KUKA KRL program: wkz7_off.src, wkz7_off.dat

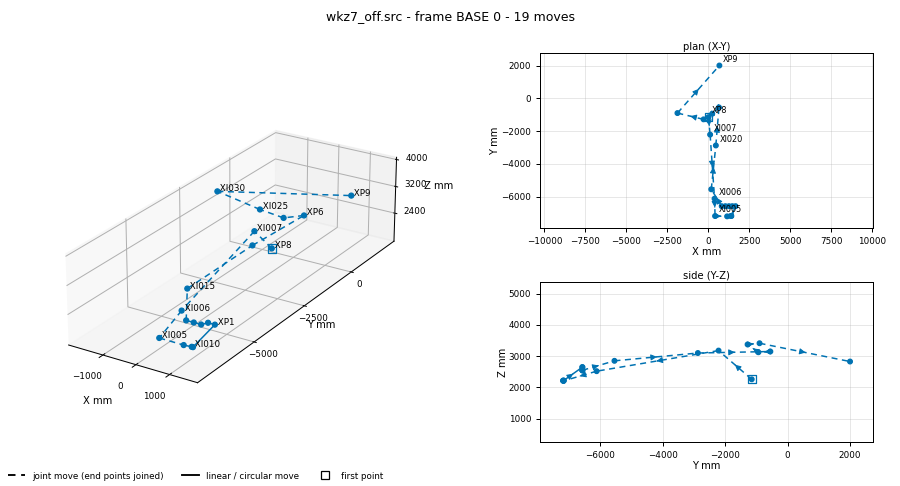
[picture p0: tool path of wkz7_off.src in frame BASE 0, 19 of 19 moves have a stored position in this frame; points joined in program order, loops and branches not executed]
--- wkz7_off.src ---
&ACCESS RVO7
&REL 553
&COMMENT Pega Gripper Axor GeoBox
&PARAM DISKPATH = KRC:\R1\Program
&PARAM TEMPLATE = C:\KRC\Roboter\Template\vorgabe
&PARAM EDITMASK = *
DEF WKZ7_OFF ( )
;FOLD INI
  ;FOLD BASISTECH INI
    GLOBAL INTERRUPT DECL 3 WHEN $STOPMESS==TRUE DO IR_STOPM ( )
    INTERRUPT ON 3
    BAS (#INITMOV,0)
  ;ENDFOLD (BASISTECH INI)
;FOLD GRIPPERTECH INI
USER_GRP(0,DUMMY,DUMMY,GDEFAULT)
;ENDFOLD (GRIPPERTECH INI)
  ;FOLD USER INI
    ;Make your modifications here

  ;ENDFOLD (USER INI)
;ENDFOLD (INI)

; Caracterizacao dos meios de producao:
; Changes: Pega Gripper na GeoBox
; Versao Atual:27/08/2015
; Name: P13.050-R2

chk_w8_wechs_ok ( )       ; CHECK TOOL CHANGE

; LIGA INTERLOCK 5 C/ R5
;FOLD Collision.Monitoring_5_On ;%{PE}%MKUKATPUSER
COLLSTOP( 5, 1 ) ;not Interrupt-Controlled
;ENDFOLD

;FOLD PTP P8 CONT Vel=100 % PDAT8 Tool[7]:Garra AXOR Base[0];%{PE}%R 8.2.20,%MKUKATPBASIS,%CMOVE,%VPTP,%P 1:PTP, 2:P8, 3:C_DIS, 5:100, 7:PDAT8
$BWDSTART=FALSE
PDAT_ACT=PPDAT8
FDAT_ACT=FP8
BAS(#PTP_PARAMS,100)
PTP XP8 C_DIS
;ENDFOLD
;FOLD PTP l007 CONT Vel=100 % P_OLP10 Tool[7]:Garra AXOR Base[0];%{PE}%R 8.2.20,%MKUKATPBASIS,%CMOVE,%VPTP,%P 1:PTP, 2:l007, 3:C_DIS, 5:100, 7:P_OLP10
$BWDSTART=FALSE
PDAT_ACT=PP_OLP10
FDAT_ACT=Fl007
BAS(#PTP_PARAMS,100)
PTP Xl007 C_DIS
;ENDFOLD
;FOLD PTP l006 CONT Vel=100 % P_OLP9 Tool[7]:Garra AXOR Base[0];%{PE}%R 8.2.20,%MKUKATPBASIS,%CMOVE,%VPTP,%P 1:PTP, 2:l006, 3:C_DIS, 5:100, 7:P_OLP9
$BWDSTART=FALSE
PDAT_ACT=PP_OLP9
FDAT_ACT=Fl006
BAS(#PTP_PARAMS,100)
PTP Xl006 C_DIS
;ENDFOLD
;FOLD PTP l005 CONT Vel=100 % P_OLP2 Tool[7]:Garra AXOR Base[0];%{PE}%R 8.2.20,%MKUKATPBASIS,%CMOVE,%VPTP,%P 1:PTP, 2:l005, 3:C_DIS, 5:100, 7:P_OLP2
$BWDSTART=FALSE
PDAT_ACT=PP_OLP2
FDAT_ACT=Fl005
BAS(#PTP_PARAMS,100)
PTP Xl005 C_DIS
;ENDFOLD
;FOLD PTP P10 Vel=100 % PDAT10 Tool[8]:Tool Changer Base[0];%{PE}%R 8.2.20,%MKUKATPBASIS,%CMOVE,%VPTP,%P 1:PTP, 2:P10, 3:, 5:100, 7:PDAT10
$BWDSTART=FALSE
PDAT_ACT=PPDAT10
FDAT_ACT=FP10
BAS(#PTP_PARAMS,100)
PTP XP10
;ENDFOLD

;FOLD OUT 3378 'Lib. p/ retirar Gripper GeoBox' State=TRUE ;%{PE}%R 8.2.20,%MKUKATPBASIS,%COUT,%VOUTX,%P 2:3378, 3:Lib. p/ retirar Gripper GeoBox, 5:TRUE, 6:
$OUT[3378]=TRUE
;ENDFOLD
;FOLD WAIT FOR ( IN 3378 'Lib. p/ retirar Gripper GeoBox' );%{PE}%R 8.2.20,%MKUKATPBASIS,%CEXT_WAIT_FOR,%VEXT_WAIT_FOR,%P 2:, 4:, 5:$IN, 6:3378, 7:Lib. p/ retirar Gripper GeoBox, 9:
WAIT FOR  ( $IN[3378] )
;ENDFOLD
;FOLD OUT 3378 'Lib. p/ retirar Gripper GeoBox' State=FALSE ;%{PE}%R 8.2.20,%MKUKATPBASIS,%COUT,%VOUTX,%P 2:3378, 3:Lib. p/ retirar Gripper GeoBox, 5:FALSE, 6:
$OUT[3378]=FALSE
;ENDFOLD
;FOLD OUT 3348 'Fora area GEOBOX' State=FALSE ;%{PE}%R 8.2.20,%MKUKATPBASIS,%COUT,%VOUTX,%P 2:3348, 3:Fora area GEOBOX, 5:FALSE, 6:
$OUT[3348]=FALSE
;ENDFOLD


;FOLD LIN l010 Vel=1 m/s CPDAT4 Tool[8]:Tool Changer Base[0];%{PE}%R 8.2.20,%MKUKATPBASIS,%CMOVE,%VLIN,%P 1:LIN, 2:l010, 3:, 5:1, 7:CPDAT4
$BWDSTART=FALSE
LDAT_ACT=LCPDAT4
FDAT_ACT=Fl010
BAS(#CP_PARAMS,1)
LIN Xl010
;ENDFOLD

;FOLD OUT 224 'Bloquear MPS' State=FALSE ;%{PE}%R 8.2.20,%MKUKATPBASIS,%COUT,%VOUTX,%P 2:224, 3:Bloquear MPS, 5:FALSE, 6:
$OUT[224]=FALSE
;ENDFOLD
;FOLD OUT 223 'Desbloquear MPS' State=TRUE ;%{PE}%R 8.2.20,%MKUKATPBASIS,%COUT,%VOUTX,%P 2:223, 3:Desbloquear MPS, 5:TRUE, 6:
$OUT[223]=TRUE
;ENDFOLD
;FOLD WAIT FOR ( IN 217 'MPS Destravado' );%{PE}%R 8.2.20,%MKUKATPBASIS,%CEXT_WAIT_FOR,%VEXT_WAIT_FOR,%P 2:, 4:, 5:$IN, 6:217, 7:MPS Destravado, 9:
WAIT FOR  ( $IN[217] )
;ENDFOLD
;FOLD WAIT FOR NOT ( IN 221 'MPS Travado' );%{PE}%R 8.2.20,%MKUKATPBASIS,%CEXT_WAIT_FOR,%VEXT_WAIT_FOR,%P 2:NOT, 4:, 5:$IN, 6:221, 7:MPS Travado, 9:
WAIT FOR  NOT ( $IN[221] )
;ENDFOLD

;FOLD ; Posicao de Pega Gripper AXOR na Geobox;%{PE}%R 8.2.20,%MKUKATPBASIS,%CCOMMENT,%VNORMAL,%P 2:Posicao de Pega Gripper  AXOR na Geobox
;ENDFOLD
;FOLD LIN P_PE11 Vel=1 m/s CPDAT6 Tool[8]:Tool Changer Base[0];%{PE}%R 8.2.20,%MKUKATPBASIS,%CMOVE,%VLIN,%P 1:LIN, 2:P_PE11, 3:, 5:1, 7:CPDAT6
$BWDSTART=FALSE
LDAT_ACT=LCPDAT6
FDAT_ACT=FP_PE11
BAS(#CP_PARAMS,1)
LIN XP_PE11
;ENDFOLD

;FOLD WAIT FOR ( IN 219 'Posicao p/ Acoplamento OK' );%{PE}%R 8.2.20,%MKUKATPBASIS,%CEXT_WAIT_FOR,%VEXT_WAIT_FOR,%P 2:, 4:, 5:$IN, 6:219, 7:Posicao p/ Acoplamento OK, 9:
WAIT FOR  ( $IN[219] )
;ENDFOLD
;FOLD OUT 223 'Desbloquear MPS' State=FALSE ;%{PE}%R 8.2.20,%MKUKATPBASIS,%COUT,%VOUTX,%P 2:223, 3:Desbloquear MPS, 5:FALSE, 6:
$OUT[223]=FALSE
;ENDFOLD
;FOLD OUT 224 'Bloquear MPS' State=TRUE ;%{PE}%R 8.2.20,%MKUKATPBASIS,%COUT,%VOUTX,%P 2:224, 3:Bloquear MPS, 5:TRUE, 6:
$OUT[224]=TRUE
;ENDFOLD
;FOLD WAIT FOR NOT ( IN 217 'MPS Destravado' );%{PE}%R 8.2.20,%MKUKATPBASIS,%CEXT_WAIT_FOR,%VEXT_WAIT_FOR,%P 2:NOT, 4:, 5:$IN, 6:217, 7:MPS Destravado, 9:
WAIT FOR  NOT ( $IN[217] )
;ENDFOLD
;FOLD WAIT FOR ( IN 221 'MPS Travado' );%{PE}%R 8.2.20,%MKUKATPBASIS,%CEXT_WAIT_FOR,%VEXT_WAIT_FOR,%P 2:, 4:, 5:$IN, 6:221, 7:MPS Travado, 9:
WAIT FOR  ( $IN[221] )
;ENDFOLD
;FOLD WAIT Time=0.5 sec;%{PE}%R 8.2.20,%MKUKATPBASIS,%CWAIT,%VWAIT,%P 3:0.5
WAIT SEC 0.5
;ENDFOLD
;FOLD IBUS ON SEGMENT_4;%{PE}%R 8.2.20,%MKUKATPBASIS,%CIBUS,%VMAP,%P 2:#ON, 3:4
$IBUS_ON=IBUS_SEGMENT[4]
$IBUS_OFF=0
;ENDFOLD
;FOLD WAIT Time=0.5 sec;%{PE}%R 8.2.20,%MKUKATPBASIS,%CWAIT,%VWAIT,%P 3:0.5
WAIT SEC 0.5
;ENDFOLD

;FOLD OUT 3379 'Lib. p/ sair c/ Gripper GeoBox' State=TRUE ;%{PE}%R 8.2.20,%MKUKATPBASIS,%COUT,%VOUTX,%P 2:3379, 3:Lib. p/ sair c/ Gripper GeoBox, 5:TRUE, 6:
$OUT[3379]=TRUE
;ENDFOLD

; ABRE GRAMPOS
;FOLD SET VACUO AXOR State=BLOW GDAT11;%{PE}%R 8.2.1,%MKUKATPGRP,%CGRP,%VGRP,%P 2:9, 4:2, 5:#NO, 6:GDAT11, 8:0, 10:0
H50(GRP,9,2,GGDAT11)
;ENDFOLD
;FOLD SET VACUO AXOR State=OFF GDAT12;%{PE}%R 8.2.1,%MKUKATPGRP,%CGRP,%VGRP,%P 2:9, 4:3, 5:#NO, 6:GDAT12, 8:0, 10:0
H50(GRP,9,3,GGDAT12)
;ENDFOLD
;FOLD SET Z2.1 RPS AXOR State=OPN GDAT25;%{PE}%R 8.2.1,%MKUKATPGRP,%CGRP,%VGRP,%P 2:10, 4:1, 5:#NO, 6:GDAT25, 8:0, 10:0
H50(GRP,10,1,GGDAT25)
;ENDFOLD
;FOLD SET Z4.1 GRP AXOR State=OPN GDAT13;%{PE}%R 8.2.1,%MKUKATPGRP,%CGRP,%VGRP,%P 2:12, 4:1, 5:#NO, 6:GDAT13, 8:0, 10:0
H50(GRP,12,1,GGDAT13)
;ENDFOLD
;FOLD SET Z5.1/2/3/4 GRP AXOR State=OPN GDAT16;%{PE}%R 8.2.1,%MKUKATPGRP,%CGRP,%VGRP,%P 2:13, 4:1, 5:#NO, 6:GDAT16, 8:0, 10:0
H50(GRP,13,1,GGDAT16)
;ENDFOLD
;FOLD SET Z6.1/2/3/4 GRP AXOR State=OPN GDAT17;%{PE}%R 8.2.1,%MKUKATPGRP,%CGRP,%VGRP,%P 2:14, 4:1, 5:#NO, 6:GDAT17, 8:0, 10:0
H50(GRP,14,1,GGDAT17)
;ENDFOLD
;FOLD SET Z7.1/2 GRP AXOR State=OPN GDAT18;%{PE}%R 8.2.1,%MKUKATPGRP,%CGRP,%VGRP,%P 2:15, 4:1, 5:#NO, 6:GDAT18, 8:0, 10:0
H50(GRP,15,1,GGDAT18)
;ENDFOLD

; VERIFICA GRAMPOS FECHADOS
chk_w7_rps2_opn( )
chk_w7_grp4_opn( )
chk_w7_grp5_opn( )
chk_w7_grp1_vacoff( )

; ABRE GRAMPO Z3.1 e VERIFICA
;FOLD SET Z3.1 GRP AXOR State=OPN GDAT26;%{PE}%R 8.2.1,%MKUKATPGRP,%CGRP,%VGRP,%P 2:11, 4:1, 5:#NO, 6:GDAT26, 8:0, 10:0
H50(GRP,11,1,GGDAT26)
;ENDFOLD
chk_w7_grp6_opn( )
chk_w7_grp7_opn( )
chk_w7_grp3_opn( )

;FOLD OUT 3379 'Solicita lib. p/ sair c/ Gripper GeoBox' State=TRUE ;%{PE}%R 8.2.20,%MKUKATPBASIS,%COUT,%VOUTX,%P 2:3379, 3:Solicita lib. p/ sair c/ Gripper GeoBox, 5:TRUE, 6:
$OUT[3379]=TRUE
;ENDFOLD
;FOLD WAIT FOR ( IN 3379 'Aguarda lib. p/ sair c/ Gripper GeoBox' );%{PE}%R 8.2.20,%MKUKATPBASIS,%CEXT_WAIT_FOR,%VEXT_WAIT_FOR,%P 2:, 4:, 5:$IN, 6:3379, 7:Aguarda lib. p/ sair c/ Gripper GeoBox, 9:
WAIT FOR  ( $IN[3379] )
;ENDFOLD
;FOLD OUT 3379 'Solicita lib. p/ sair c/ Gripper GeoBox' State=FALSE ;%{PE}%R 8.2.20,%MKUKATPBASIS,%COUT,%VOUTX,%P 2:3379, 3:Solicita lib. p/ sair c/ Gripper GeoBox, 5:FALSE, 6:
$OUT[3379]=FALSE
;ENDFOLD

;FOLD LIN P1 CONT Vel=1 m/s CPDAT2 Tool[7]:Garra AXOR Base[0];%{PE}%R 8.2.20,%MKUKATPBASIS,%CMOVE,%VLIN,%P 1:LIN, 2:P1, 3:C_DIS C_DIS, 5:1, 7:CPDAT2
$BWDSTART=FALSE
LDAT_ACT=LCPDAT2
FDAT_ACT=FP1
BAS(#CP_PARAMS,1)
LIN XP1 C_DIS C_DIS
;ENDFOLD
;FOLD LIN P3 CONT Vel=1 m/s CPDAT5 Tool[7]:Garra AXOR Base[0];%{PE}%R 8.2.20,%MKUKATPBASIS,%CMOVE,%VLIN,%P 1:LIN, 2:P3, 3:C_DIS C_DIS, 5:1, 7:CPDAT5
$BWDSTART=FALSE
LDAT_ACT=LCPDAT5
FDAT_ACT=FP3
BAS(#CP_PARAMS,1)
LIN XP3 C_DIS C_DIS
;ENDFOLD

;FOLD LIN P14 Vel=1 m/s CPDAT9 Tool[7]:Garra AXOR Base[0];%{PE}%R 8.2.20,%MKUKATPBASIS,%CMOVE,%VLIN,%P 1:LIN, 2:P14, 3:, 5:1, 7:CPDAT9
$BWDSTART=FALSE
LDAT_ACT=LCPDAT9
FDAT_ACT=FP14
BAS(#CP_PARAMS,1)
LIN XP14
;ENDFOLD

;FOLD PULSE 3335 'R2 retirou garra da Geo' State=TRUE Time=3 sec;%{PE}%R 8.2.20,%MKUKATPBASIS,%COUT,%VPULSE,%P 2:3335, 3:R2 retirou garra da Geo, 5:TRUE, 6:, 8:3
PULSE($OUT[3335], TRUE,3)
;ENDFOLD

;FOLD PTP P13 CONT Vel=100 % PDAT12 Tool[7]:Garra AXOR Base[0];%{PE}%R 8.2.20,%MKUKATPBASIS,%CMOVE,%VPTP,%P 1:PTP, 2:P13, 3:C_DIS, 5:100, 7:PDAT12
$BWDSTART=FALSE
PDAT_ACT=PPDAT12
FDAT_ACT=FP13
BAS(#PTP_PARAMS,100)
PTP XP13 C_DIS
;ENDFOLD

; DESLIGA INTERLOCK 5 C/ R5
;FOLD Collision.Monitoring_5_Off . ;%{PE}%MKUKATPUSER
COLLSTOP( 5, 2+0 )
;ENDFOLD

;FOLD PTP P11 CONT Vel=100 % PDAT13 Tool[7]:Garra AXOR Base[0];%{PE}%R 8.2.20,%MKUKATPBASIS,%CMOVE,%VPTP,%P 1:PTP, 2:P11, 3:C_DIS, 5:100, 7:PDAT13
$BWDSTART=FALSE
PDAT_ACT=PPDAT13
FDAT_ACT=FP11
BAS(#PTP_PARAMS,100)
PTP XP11 C_DIS
;ENDFOLD
;FOLD PTP l015 CONT Vel=100 % PDAT4 Tool[7]:Garra AXOR Base[0];%{PE}%R 8.2.20,%MKUKATPBASIS,%CMOVE,%VPTP,%P 1:PTP, 2:l015, 3:C_DIS, 5:100, 7:PDAT4
$BWDSTART=FALSE
PDAT_ACT=PPDAT4
FDAT_ACT=Fl015
BAS(#PTP_PARAMS,100)
PTP Xl015 C_DIS
;ENDFOLD
;FOLD PTP l020 CONT Vel=100 % P_OLP4 Tool[7]:Garra AXOR Base[0];%{PE}%R 8.2.20,%MKUKATPBASIS,%CMOVE,%VPTP,%P 1:PTP, 2:l020, 3:C_DIS, 5:100, 7:P_OLP4
$BWDSTART=FALSE
PDAT_ACT=PP_OLP4
FDAT_ACT=Fl020
BAS(#PTP_PARAMS,100)
PTP Xl020 C_DIS
;ENDFOLD
;FOLD PTP P6 CONT Vel=100 % PDAT6 Tool[7]:Garra AXOR Base[0];%{PE}%R 8.2.20,%MKUKATPBASIS,%CMOVE,%VPTP,%P 1:PTP, 2:P6, 3:C_DIS, 5:100, 7:PDAT6
$BWDSTART=FALSE
PDAT_ACT=PPDAT6
FDAT_ACT=FP6
BAS(#PTP_PARAMS,100)
PTP XP6 C_DIS
;ENDFOLD

;FOLD WAIT FOR ( IN 190 'DOCK 4 Proteção Fechada' ) CONT;%{PE}%R 8.2.20,%MKUKATPBASIS,%CEXT_WAIT_FOR,%VEXT_WAIT_FOR,%P 2:, 4:, 5:$IN, 6:190, 7:DOCK 4 Proteção Fechada, 9:CONTINUE
CONTINUE
WAIT FOR  ( $IN[190] )
;ENDFOLD
;FOLD WAIT FOR ( IN 198 'DOCK 5 Proteção Fechada' ) CONT;%{PE}%R 8.2.20,%MKUKATPBASIS,%CEXT_WAIT_FOR,%VEXT_WAIT_FOR,%P 2:, 4:, 5:$IN, 6:198, 7:DOCK 5 Proteção Fechada, 9:CONTINUE
CONTINUE
WAIT FOR  ( $IN[198] )
;ENDFOLD

;FOLD OUT 3348 'Fora area GEOBOX' State=TRUE ;%{PE}%R 8.2.20,%MKUKATPBASIS,%COUT,%VOUTX,%P 2:3348, 3:Fora area GEOBOX, 5:TRUE, 6:
$OUT[3348]=TRUE
;ENDFOLD

;FOLD PTP P7 CONT Vel=100 % PDAT7 Tool[7]:Garra AXOR Base[0];%{PE}%R 8.2.20,%MKUKATPBASIS,%CMOVE,%VPTP,%P 1:PTP, 2:P7, 3:C_DIS, 5:100, 7:PDAT7
$BWDSTART=FALSE
PDAT_ACT=PPDAT7
FDAT_ACT=FP7
BAS(#PTP_PARAMS,100)
PTP XP7 C_DIS
;ENDFOLD

; FECHA GRAMPOS GARRA AXOR
;FOLD SET Z3.1 GRP AXOR State=CLO CONT at START Delay=1 ms;%{PE}%R 8.2.1,%MKUKATPGRP,%CGRP,%VGRP,%P 2:11, 4:2, 5:#YES, 6:GDAT19, 8:0, 10:1
TRIGGER WHEN DISTANCE=0 DELAY=1 DO H50(GRP_APO,11,2,GCONT) PRIO=-1
;ENDFOLD
;FOLD SET Z4.1 GRP AXOR State=CONT at START Delay=1 ms;%{PE}%R 8.2.1,%MKUKATPGRP,%CGRP,%VGRP,%P 2:12, 4:2, 5:#YES, 6:GDAT20, 8:0, 10:1
TRIGGER WHEN DISTANCE=0 DELAY=1 DO H50(GRP_APO,12,2,GCONT) PRIO=-1
;ENDFOLD
;FOLD SET Z5.1/2/3/4 GRP AXOR State=CLO CONT at START Delay=1 ms;%{PE}%R 8.2.1,%MKUKATPGRP,%CGRP,%VGRP,%P 2:13, 4:2, 5:#YES, 6:GDAT21, 8:0, 10:1
TRIGGER WHEN DISTANCE=0 DELAY=1 DO H50(GRP_APO,13,2,GCONT) PRIO=-1
;ENDFOLD
;FOLD SET Z6.1/2/3/4 GRP AXOR State=CLO CONT at START Delay=1 ms;%{PE}%R 8.2.1,%MKUKATPGRP,%CGRP,%VGRP,%P 2:14, 4:2, 5:#YES, 6:GDAT22, 8:0, 10:1
TRIGGER WHEN DISTANCE=0 DELAY=1 DO H50(GRP_APO,14,2,GCONT) PRIO=-1
;ENDFOLD
;FOLD SET Z7.1/2 GRP AXOR State=CLO CONT at START Delay=1 ms;%{PE}%R 8.2.1,%MKUKATPGRP,%CGRP,%VGRP,%P 2:15, 4:2, 5:#YES, 6:GDAT23, 8:0, 10:1
TRIGGER WHEN DISTANCE=0 DELAY=1 DO H50(GRP_APO,15,2,GCONT) PRIO=-1
;ENDFOLD

;FOLD PTP l025 CONT Vel=100 % P_OLP5 Tool[7]:Garra AXOR Base[0];%{PE}%R 8.2.20,%MKUKATPBASIS,%CMOVE,%VPTP,%P 1:PTP, 2:l025, 3:C_DIS, 5:100, 7:P_OLP5
$BWDSTART=FALSE
PDAT_ACT=PP_OLP5
FDAT_ACT=Fl025
BAS(#PTP_PARAMS,100)
PTP Xl025 C_DIS
;ENDFOLD
;FOLD PTP l030 CONT Vel=100 % P_OLP6 Tool[7]:Garra AXOR Base[0];%{PE}%R 8.2.20,%MKUKATPBASIS,%CMOVE,%VPTP,%P 1:PTP, 2:l030, 3:C_DIS, 5:100, 7:P_OLP6
$BWDSTART=FALSE
PDAT_ACT=PP_OLP6
FDAT_ACT=Fl030
BAS(#PTP_PARAMS,100)
PTP Xl030 C_DIS
;ENDFOLD
;FOLD PTP P9 CONT Vel=100 % PDAT9 Tool[7]:Garra AXOR Base[0];%{PE}%R 8.2.20,%MKUKATPBASIS,%CMOVE,%VPTP,%P 1:PTP, 2:P9, 3:C_DIS, 5:100, 7:PDAT9
$BWDSTART=FALSE
PDAT_ACT=PPDAT9
FDAT_ACT=FP9
BAS(#PTP_PARAMS,100)
PTP XP9 C_DIS
;ENDFOLD

END

--- wkz7_off.dat ---
&ACCESS RVO7
&REL 553
&COMMENT Pega Gripper Axor GeoBox
&PARAM DISKPATH = KRC:\R1\Program
&PARAM TEMPLATE = C:\KRC\Roboter\Template\vorgabe
&PARAM EDITMASK = *
DEFDAT  wkz7_off
;FOLD EXTERNAL DECLARATIONS;%{PE}%MKUKATPBASIS,%CEXT,%VCOMMON,%P
;FOLD GRIPPERTECH EXT
EXT  H50 (INT  :IN,INT  :IN,INT  :IN,GRP_TYP  :IN )
;ENDFOLD (GRIPPERTECH EXT)
;FOLD SPOTTECH EXT
EXT  USERSPOT (S_COMMAND  :IN,SPOT_TYPE  :IN )
;ENDFOLD (SPOTTECH EXT)
;FOLD BASISTECH EXT;%{PE}%MKUKATPBASIS,%CEXT,%VEXT,%P
EXT  BAS (BAS_COMMAND  :IN,REAL  :IN )
DECL INT SUCCESS
;ENDFOLD (BASISTECH EXT)
;FOLD USER EXT;%{E}%MKUKATPUSER,%CEXT,%VEXT,%P
;Make your modifications here

INT Dep_ocup
INT Prot_Ab
INT Prot_Fech
INT Abrir_Prot
INT Fechar_Prot
INT Segmento

;ENDFOLD (USER EXT)
;ENDFOLD (EXTERNAL DECLARATIONS)
DECL FDAT FLX1741={TOOL_NO 8,BASE_NO 0,IPO_FRAME #BASE,POINT2[] " "}
DECL PDAT PP_OLP1={VEL 100.0,ACC 100.0,APO_DIST 0.0}
DECL FDAT Fl005={TOOL_NO 8,BASE_NO 0,IPO_FRAME #BASE,POINT2[] " "}
DECL PDAT PP_OLP2={VEL 100.0,ACC 100.0,APO_DIST 100.0,APO_MODE #CDIS}
DECL E6POS Xl005={X 403.914795,Y -7174.31689,Z 2205.16992,A 90.3375092,B -44.8243294,C 89.1014404,S 2,T 42,E1 -4904.96777,E2 0.0,E3 0.0,E4 0.0,E5 0.0,E6 0.0}
DECL FDAT Fl010={TOOL_NO 8,BASE_NO 0,IPO_FRAME #BASE,POINT2[] " "}
DECL PDAT PP_OLP3={VEL 100.0,ACC 100.0,APO_DIST 0.0}
DECL E6POS Xl010={X 1360.66199,Y -7173.98389,Z 2215.25098,A 90.3056412,B -44.8249512,C 89.3882599,S 2,T 43,E1 -4904.96777,E2 0.0,E3 0.0,E4 0.0,E5 0.0,E6 0.0}
DECL FDAT FP_PE11={TOOL_NO 8,BASE_NO 0,IPO_FRAME #BASE,POINT2[] " ",TQ_STATE FALSE}
DECL E6POS XP_PE11={X 1396.64404,Y -7173.98779,Z 2215.24292,A 90.3045883,B -44.8244591,C 89.3893127,S 2,T 43,E1 -4904.96924,E2 0.0,E3 0.0,E4 0.0,E5 0.0,E6 0.0}
DECL LDAT LL_OLP1={VEL 0.25,ACC 100.0,APO_DIST 0.0,APO_FAC 0.0,ORI_TYP #VAR,CIRC_TYP #BASE,JERK_FAC 50.0}
DECL FDAT Fl015={TOOL_NO 7,BASE_NO 0,IPO_FRAME #BASE,POINT2[] " ",TQ_STATE FALSE}
DECL E6POS Xl015={X 171.100998,Y -5544.98486,Z 2848.19995,A -27.08494,B 89.5359268,C -96.8980103,S 2,T 42,E1 -4008.10303,E2 0.0,E3 0.0,E4 0.0,E5 0.0,E6 0.0}
DECL LDAT LL_OLP2={VEL 0.25,ACC 100.0,APO_DIST 0.0,APO_FAC 0.0,ORI_TYP #VAR,CIRC_TYP #BASE,JERK_FAC 50.0}
DECL FDAT Fl020={TOOL_NO 7,BASE_NO 0,IPO_FRAME #BASE,POINT2[] " ",TQ_STATE FALSE}
DECL PDAT PP_OLP4={VEL 100.0,ACC 100.0,APO_DIST 100.0,APO_MODE #CDIS}
DECL E6POS Xl020={X 450.387299,Y -2873.21899,Z 3097.83008,A -106.307198,B 76.5619431,C -152.027603,S 2,T 42,E1 -1270.07397,E2 0.0,E3 0.0,E4 0.0,E5 0.0,E6 0.0}
DECL FDAT Fl025={TOOL_NO 7,BASE_NO 0,IPO_FRAME #BASE,POINT2[] " ",TQ_STATE FALSE}
DECL PDAT PP_OLP5={VEL 100.0,ACC 100.0,APO_DIST 100.0,APO_MODE #CDIS}
DECL E6POS Xl025={X -297.052795,Y -1281.25305,Z 3372.53589,A -143.016907,B 70.3474884,C -128.409393,S 2,T 42,E1 393.984894,E2 0.0,E3 0.0,E4 0.0,E5 0.0,E6 0.0}
DECL FDAT Fl030={TOOL_NO 7,BASE_NO 0,IPO_FRAME #BASE,POINT2[] " ",TQ_STATE FALSE}
DECL PDAT PP_OLP6={VEL 100.0,ACC 100.0,APO_DIST 100.0,APO_MODE #CDIS}
DECL E6POS Xl030={X -1889.92395,Y -898.348389,Z 3411.10498,A 45.4453201,B 85.3523483,C 155.626099,S 2,T 34,E1 -248.645798,E2 0.0,E3 0.0,E4 0.0,E5 0.0,E6 0.0}
DECL FDAT Fl035={TOOL_NO 7,BASE_NO 0,IPO_FRAME #BASE,POINT2[] " "}
DECL PDAT PP_OLP7={VEL 100.0,ACC 100.0,APO_DIST 0.0}
DECL E6POS Xl035={X 250.487,Y -7591.85303,Z 1923.70703,A -24.4409008,B -89.4464035,C 109.612,S 2,T 42,E1 -4700.0,E2 0.0,E3 0.0,E4 0.0,E5 0.0,E6 0.0}
DECL FDAT FLX1710={TOOL_NO 7,BASE_NO 0,IPO_FRAME #BASE,POINT2[] " "}
DECL PDAT PP_OLP8={VEL 100.0,ACC 100.0,APO_DIST 0.0}
DECL BASIS_SUGG_T LAST_BASIS={POINT1[] "P15                     ",POINT2[] "P15                     ",CP_PARAMS[] "CPDAT9                  ",PTP_PARAMS[] "PDAT14                  ",CONT[] "                        ",CP_VEL[] "1                       ",PTP_VEL[] "100                     ",SYNC_PARAMS[] "SYNCDAT                 ",SPL_NAME[] "S0                      "}
DECL PDAT PP_OLP9={VEL 100.0,ACC 100.0,APO_DIST 100.0,APO_MODE #CDIS}
DECL E6POS Xl006={X 371.434387,Y -6115.61182,Z 2516.23511,A 38.8590508,B -48.6963615,C 119.477798,S 2,T 42,E1 -4092.36304,E2 0.0,E3 0.0,E4 0.0,E5 0.0,E6 0.0}
DECL FDAT Fl006={TOOL_NO 8,BASE_NO 0,IPO_FRAME #BASE,POINT2[] " ",TQ_STATE FALSE}
DECL PDAT PP_OLP10={VEL 100.0,ACC 100.0,APO_DIST 100.0,APO_MODE #CDIS}
DECL E6POS Xl007={X 101.848396,Y -2211.33911,Z 3175.94702,A 55.6541481,B -26.1408596,C 89.2244034,S 2,T 42,E1 -694.004272,E2 0.0,E3 0.0,E4 0.0,E5 0.0,E6 0.0}
DECL FDAT Fl007={TOOL_NO 8,BASE_NO 0,IPO_FRAME #BASE,POINT2[] " "}
DECL PDAT PP_OLP11={VEL 100.0,ACC 100.0,APO_DIST 0.0}
DECL E6POS Xl008={X -575.517883,Y -1850.71594,Z 3336.90405,A -36.2922897,B -43.9408302,C 86.1404572,S 2,T 42,E1 -1386.47595,E2 0.0,E3 0.0,E4 0.0,E5 0.0,E6 0.0}
DECL FDAT Fl008={TOOL_NO 8,BASE_NO 0,IPO_FRAME #BASE,POINT2[] " "}
DECL PDAT PPDAT1={VEL 100.0,ACC 100.0,APO_DIST 100.0}
DECL LDAT LCPDAT1={VEL 2.0,ACC 100.0,APO_DIST 100.0,APO_FAC 50.0,AXIS_VEL 100.0,AXIS_ACC 100.0,ORI_TYP #VAR,CIRC_TYP #BASE,JERK_FAC 50.0,GEAR_JERK 50.0,EXAX_IGN 0}
DECL LDAT LCPDAT0={VEL 2.0,ACC 100.0,APO_DIST 100.0,APO_FAC 50.0,AXIS_VEL 100.0,AXIS_ACC 100.0,ORI_TYP #VAR,CIRC_TYP #BASE,JERK_FAC 50.0,GEAR_JERK 50.0,EXAX_IGN 0}
DECL E6POS XP0={X 1395.83496,Y -7173.34619,Z 2283.36499,A 90.5466232,B -44.6719093,C 89.2932816,S 2,T 43,E1 -5561.28906,E2 0.0,E3 0.0,E4 0.0,E5 0.0,E6 0.0}
DECL FDAT FP0={TOOL_NO 8,BASE_NO 0,IPO_FRAME #BASE,POINT2[] " ",TQ_STATE FALSE}
DECL PDAT PPDAT2={VEL 100.0,ACC 100.0,APO_DIST 100.0}
DECL PDAT PPDAT3={VEL 100.0,ACC 100.0,APO_DIST 100.0}
DECL E6POS XP1={X 1651.76294,Y -6573.12207,Z 2645.26196,A -22.0089207,B 89.5332031,C -96.8824005,S 2,T 43,E1 -4904.96777,E2 0.0,E3 0.0,E4 0.0,E5 0.0,E6 0.0}
DECL FDAT FP1={TOOL_NO 7,BASE_NO 0,IPO_FRAME #BASE,POINT2[] " ",TQ_STATE FALSE}
DECL LDAT LCPDAT2={VEL 2.0,ACC 100.0,APO_DIST 100.0,APO_FAC 50.0,AXIS_VEL 100.0,AXIS_ACC 100.0,ORI_TYP #VAR,CIRC_TYP #BASE,JERK_FAC 50.0,GEAR_JERK 50.0,EXAX_IGN 0}
DECL E6POS XP2={X 855.30658,Y -6573.16699,Z 2645.25098,A -22.0339794,B 89.5358429,C -96.905899,S 2,T 43,E1 -4904.96777,E2 0.0,E3 0.0,E4 0.0,E5 0.0,E6 0.0}
DECL FDAT FP2={TOOL_NO 10,BASE_NO 0,IPO_FRAME #BASE,POINT2[] " ",TQ_STATE FALSE}
DECL LDAT LCPDAT3={VEL 2.0,ACC 100.0,APO_DIST 100.0,APO_FAC 50.0,AXIS_VEL 100.0,AXIS_ACC 100.0,ORI_TYP #VAR,CIRC_TYP #BASE,JERK_FAC 50.0,GEAR_JERK 50.0,EXAX_IGN 0}
DECL LDAT LCPDAT4={VEL 2.0,ACC 100.0,APO_DIST 100.0,APO_FAC 50.0,AXIS_VEL 100.0,AXIS_ACC 100.0,ORI_TYP #VAR,CIRC_TYP #BASE,JERK_FAC 50.0,GEAR_JERK 50.0,EXAX_IGN 0}
DECL GRP_SUGG_T LAST_GRP={NUMBER[] "9                       ",STATE[] "3                       ",PARAMS[] "GDAT10                  "}
DECL GRP_TYP GGDAT1={G_APO #NO,GRP_TIME 0.200000003,CTRL #OFF,DLY 0,DST 1}
DECL GRP_TYP GGDAT2={G_APO #NO,GRP_TIME 0.200000003,CTRL #OFF,DLY 0,DST 1}
DECL GRP_TYP GGDAT3={G_APO #NO,GRP_TIME 0.200000003,CTRL #OFF,DLY 0,DST 1}
DECL GRP_TYP GGDAT4={G_APO #NO,GRP_TIME 0.200000003,CTRL #OFF,DLY 0,DST 1}
DECL GRP_TYP GGDAT5={G_APO #NO,GRP_TIME 0.200000003,CTRL #OFF,DLY 0,DST 1}
DECL GRP_TYP GGDAT6={G_APO #NO,GRP_TIME 0.200000003,CTRL #OFF,DLY 0,DST 1}
DECL GRP_TYP GGDAT7={G_APO #NO,GRP_TIME 0.200000003,CTRL #OFF,DLY 0,DST 1}
DECL GRP_TYP GGDAT8={G_APO #NO,GRP_TIME 0.200000003,CTRL #OFF,DLY 0,DST 1}
DECL E6POS XP3={X 1452.60205,Y -6573.13721,Z 2645.26196,A -21.9808407,B 89.5339127,C -96.8539276,S 2,T 43,E1 -4904.96777,E2 0.0,E3 0.0,E4 0.0,E5 0.0,E6 0.0}
DECL FDAT FP3={TOOL_NO 7,BASE_NO 0,IPO_FRAME #BASE,POINT2[] " ",TQ_STATE FALSE}
DECL LDAT LCPDAT5={VEL 2.0,ACC 100.0,APO_DIST 100.0,APO_FAC 50.0,AXIS_VEL 100.0,AXIS_ACC 100.0,ORI_TYP #VAR,CIRC_TYP #BASE,JERK_FAC 50.0,GEAR_JERK 50.0,EXAX_IGN 0}
DECL PDAT PPDAT4={VEL 100.0,ACC 100.0,APO_DIST 100.0,APO_MODE #CDIS}
DECL PDAT PPDAT0={VEL 100.0,ACC 100.0,APO_DIST 100.0}
DECL E6POS XP4={X -215.321304,Y 1293.63403,Z 2633.10791,A 73.3692017,B 61.8229599,C -101.250298,S 2,T 34,E1 -367.387085,E2 0.0,E3 0.0,E4 0.0,E5 0.0,E6 0.0}
DECL FDAT FP4={TOOL_NO 7,BASE_NO 0,IPO_FRAME #BASE,POINT2[] " ",TQ_STATE FALSE}
DECL E6POS XP5={X 972.294128,Y 190.753998,Z 773.197021,A -179.483704,B 59.8206406,C 90.6673584,S 2,T 43,E1 -4904.96777,E2 0.0,E3 0.0,E4 0.0,E5 0.0,E6 0.0}
DECL FDAT FP5={TOOL_NO 7,BASE_NO 3,IPO_FRAME #BASE,POINT2[] " ",TQ_STATE FALSE}
DECL PDAT PPDAT5={VEL 100.0,ACC 100.0,APO_DIST 100.0}
DECL LDAT LCPDAT6={VEL 2.0,ACC 100.0,APO_DIST 100.0,APO_FAC 50.0,AXIS_VEL 100.0,AXIS_ACC 100.0,ORI_TYP #VAR,CIRC_TYP #BASE,JERK_FAC 50.0,GEAR_JERK 50.0,EXAX_IGN 0}
DECL E6POS XP6={X 641.568115,Y -551.410583,Z 3146.56689,A -106.381897,B 74.4718018,C -152.111801,S 2,T 42,E1 415.521912,E2 0.0,E3 0.0,E4 0.0,E5 0.0,E6 0.0}
DECL FDAT FP6={TOOL_NO 7,BASE_NO 0,IPO_FRAME #BASE,POINT2[] " ",TQ_STATE FALSE}
DECL PDAT PPDAT6={VEL 100.0,ACC 100.0,APO_DIST 100.0,APO_MODE #CDIS}
DECL E6POS XP7={X 233.5112,Y -934.783386,Z 3122.1731,A -135.993805,B 77.6455307,C -139.065399,S 2,T 42,E1 400.201904,E2 0.0,E3 0.0,E4 0.0,E5 0.0,E6 0.0}
DECL FDAT FP7={TOOL_NO 7,BASE_NO 0,IPO_FRAME #BASE,POINT2[] " ",TQ_STATE FALSE}
DECL PDAT PPDAT7={VEL 100.0,ACC 100.0,APO_DIST 100.0,APO_MODE #CDIS}
DECL GRP_TYP GGDAT9={G_APO #NO,GRP_TIME 0.200000003,CTRL #OFF,DLY 0,DST 1}
DECL GRP_TYP GGDAT10={G_APO #NO,GRP_TIME 0.200000003,CTRL #OFF,DLY 0,DST 1}
DECL GRP_TYP GGDAT11={G_APO #NO,GRP_TIME 0.200000003,CTRL #OFF,DLY 0,DST 1}
DECL GRP_TYP GGDAT12={G_APO #NO,GRP_TIME 0.200000003,CTRL #OFF,DLY 0,DST 1}
DECL GRP_TYP GGDAT13={G_APO #NO,GRP_TIME 0.200000003,CTRL #OFF,DLY 0,DST 1}
DECL GRP_TYP GGDAT14={G_APO #NO,GRP_TIME 0.200000003,CTRL #OFF,DLY 0,DST 1}
DECL GRP_TYP GGDAT15={G_APO #NO,GRP_TIME 0.200000003,CTRL #OFF,DLY 0,DST 1}
DECL GRP_TYP GGDAT16={G_APO #NO,GRP_TIME 0.200000003,CTRL #OFF,DLY 0,DST 1}
DECL GRP_TYP GGDAT17={G_APO #NO,GRP_TIME 0.200000003,CTRL #OFF,DLY 0,DST 1}
DECL GRP_TYP GGDAT18={G_APO #NO,GRP_TIME 0.200000003,CTRL #OFF,DLY 0,DST 1}
DECL GRP_TYP GGDAT19={G_APO #NO,GRP_TIME 0.200000003,CTRL #OFF,DLY 0,DST 1}
DECL GRP_TYP GGDAT20={G_APO #NO,GRP_TIME 0.200000003,CTRL #OFF,DLY 0,DST 1}
DECL GRP_TYP GGDAT21={G_APO #NO,GRP_TIME 0.200000003,CTRL #OFF,DLY 0,DST 1}
DECL GRP_TYP GGDAT22={G_APO #NO,GRP_TIME 0.200000003,CTRL #OFF,DLY 0,DST 1}
DECL GRP_TYP GGDAT23={G_APO #NO,GRP_TIME 0.200000003,CTRL #OFF,DLY 0,DST 1}
DECL GRP_TYP GCONT={G_APO #YES,GRP_TIME 0.0,CTRL #OFF,DLY 0,DST 0}
DECL GRP_TYP GGDAT24={G_APO #NO,GRP_TIME 0.200000003,CTRL #OFF,DLY 0,DST 1}
DECL E6POS XP8={X 0.000957992917,Y -1148.60498,Z 2255.92505,A 103.8032,B 19.4667301,C -175.319504,S 2,T 10,E1 200.000198,E2 0.0,E3 0.0,E4 0.0,E5 0.0,E6 0.0}
DECL FDAT FP8={TOOL_NO 8,BASE_NO 0,IPO_FRAME #BASE,POINT2[] " ",TQ_STATE FALSE}
DECL PDAT PPDAT8={VEL 100.0,ACC 100.0,APO_DIST 100.0,APO_MODE #CDIS}
DECL E6POS XP9={X 666.23822,Y 2000.17297,Z 2825.34399,A -88.6034088,B -68.5179062,C -78.75,S 6,T 50,E1 387.465515,E2 0.0,E3 0.0,E4 0.0,E5 0.0,E6 0.0}
DECL FDAT FP9={TOOL_NO 7,BASE_NO 0,IPO_FRAME #BASE,POINT2[] " ",TQ_STATE FALSE}
DECL PDAT PPDAT9={VEL 100.0,ACC 100.0,APO_DIST 100.0,APO_MODE #CDIS}
DECL E6POS XP10={X 1138.20996,Y -7194.12012,Z 2212.39502,A 90.0621872,B -44.7253799,C 89.709877,S 2,T 43,E1 -4904.96777,E2 0.0,E3 0.0,E4 0.0,E5 0.0,E6 0.0}
DECL FDAT FP10={TOOL_NO 8,BASE_NO 0,IPO_FRAME #BASE,POINT2[] " ",TQ_STATE FALSE}
DECL PDAT PPDAT10={VEL 100.0,ACC 100.0,APO_DIST 100.0}
DECL GRP_TYP GGDAT25={G_APO #NO,GRP_TIME 0.200000003,CTRL #OFF,DLY 0,DST 1}
DECL GRP_TYP GGDAT26={G_APO #NO,GRP_TIME 0.200000003,CTRL #OFF,DLY 0,DST 1}
DECL E6POS XP11={X 807.894775,Y -6573.12695,Z 2544.31812,A -178.418503,B 83.6518021,C 106.697701,S 2,T 42,E1 -4904.96777,E2 0.0,E3 0.0,E4 0.0,E5 0.0,E6 0.0}
DECL FDAT FP11={TOOL_NO 7,BASE_NO 0,IPO_FRAME #BASE,POINT2[] " ",TQ_STATE FALSE}
DECL LDAT LCPDAT7={VEL 2.0,ACC 100.0,APO_DIST 100.0,APO_FAC 50.0,AXIS_VEL 100.0,AXIS_ACC 100.0,ORI_TYP #VAR,CIRC_TYP #BASE,JERK_FAC 50.0,GEAR_JERK 50.0,EXAX_IGN 0}
DECL E6POS XP12={X 1290.94604,Y -6573.13623,Z 2544.33911,A -178.421295,B 83.6524429,C 106.695297,S 2,T 43,E1 -4904.96777,E2 0.0,E3 0.0,E4 0.0,E5 0.0,E6 0.0}
DECL FDAT FP12={TOOL_NO 10,BASE_NO 0,IPO_FRAME #BASE,POINT2[] " ",TQ_STATE FALSE}
DECL PDAT PPDAT11={VEL 100.0,ACC 100.0,APO_DIST 50.0,APO_MODE #CDIS}
DECL E6POS XP13={X 1032.25403,Y -6573.13281,Z 2544.33008,A -178.4207,B 83.6519775,C 106.695602,S 2,T 43,E1 -4904.96777,E2 0.0,E3 0.0,E4 0.0,E5 0.0,E6 0.0}
DECL FDAT FP13={TOOL_NO 7,BASE_NO 0,IPO_FRAME #BASE,POINT2[] " ",TQ_STATE FALSE}
DECL PDAT PPDAT12={VEL 100.0,ACC 100.0,APO_DIST 100.0,APO_MODE #CDIS}
DECL LDAT LCPDAT8={VEL 2.0,ACC 100.0,APO_DIST 50.0,APO_FAC 50.0,AXIS_VEL 100.0,AXIS_ACC 100.0,ORI_TYP #VAR,CIRC_TYP #BASE,JERK_FAC 50.0,GEAR_JERK 50.0,EXAX_IGN 0}
DECL E6POS XP14={X 1249.51599,Y -6573.13818,Z 2544.33911,A -178.421402,B 83.6520767,C 106.695099,S 2,T 43,E1 -4904.96777,E2 0.0,E3 0.0,E4 0.0,E5 0.0,E6 0.0}
DECL FDAT FP14={TOOL_NO 7,BASE_NO 0,IPO_FRAME #BASE,POINT2[] " ",TQ_STATE FALSE}
DECL LDAT LCPDAT9={VEL 2.0,ACC 100.0,APO_DIST 100.0,APO_FAC 50.0,AXIS_VEL 100.0,AXIS_ACC 100.0,ORI_TYP #VAR,CIRC_TYP #BASE,JERK_FAC 50.0,GEAR_JERK 50.0,EXAX_IGN 0}
DECL PDAT PPDAT13={VEL 100.0,ACC 100.0,APO_DIST 100.0,APO_MODE #CDIS}
DECL E6POS XP15={X 1708.40503,Y -6573.14307,Z 2638.80298,A -22.0332108,B 89.5358124,C -96.9054565,S 2,T 43,E1 -4904.96289,E2 0.0,E3 0.0,E4 0.0,E5 0.0,E6 0.0}
DECL FDAT FP15={TOOL_NO 7,BASE_NO 0,IPO_FRAME #BASE,POINT2[] " ",TQ_STATE FALSE}
DECL PDAT PPDAT14={VEL 100.0,ACC 100.0,APO_DIST 100.0}
ENDDAT
